FUNCTION_BLOCK fb_Camming
VAR
  _ItfAxisSlave   : I_McAxis;
  _ItfAxisMaster  : I_McAxis;

    
END_VAR

END_FUNCTION_BLOCK

(* stored: Version 1.1.0.1, ProductVersion 3.1.4024.12
   POU fb_Camming: Id {527605ca-3a86-0df1-134f-058287ba4975}, SpecialFunc None *)
